(* IEC 61131-3 sources: ATCMcontrol_Engineering/src/Target/ATHW119/Libs/HW119, 8 files *)

(* ---- HW119_CloseCrossTable.st ---- *)
(*[[
    UserText1= "hw119_close_cross_table",
    UserHelpURL= "ATCMfile:HW119_CloseCrossTable.HTML",
]]*)
FUNCTION HW119_CloseCrossTable : UINT
VAR_INPUT
END_VAR
INLINE {STDLIB(HW119_CloseCrossTable)}
END_FUNCTION

(* ---- HW119_dword2float.st ---- *)
(*[[
    UserHelpURL= "ATCMfile:HW119_dword2float.HTML",
    UserText1= "HW119_dword2float",
]]*)
FUNCTION HW119_dword2float : REAL
VAR_INPUT
    dwordvalue : DWORD; (*[dword value to convert]*)
END_VAR
INLINE {STDLIB(HW119_dword2float)}
END_FUNCTION

(* ---- HW119_float2dword.st ---- *)
(*[[
    UserHelpURL= "ATCMfile:HW119_float2dword.HTML",
    UserText1= "HW119_float2dword",
]]*)
FUNCTION HW119_float2dword : DWORD
VAR_INPUT
    realvalue : REAL; (*[float value to convert]*)
END_VAR
INLINE {STDLIB(HW119_float2dword)}
END_FUNCTION

(* ---- HW119_GetAddr.st ---- *)
(*[[
    UserText1= "hw119_get_addr",
    UserHelpURL= "ATCMfile:HW119_GetAddr.HTML",
]]*)
FUNCTION HW119_GetAddr : WORD
VAR_INPUT
    varname : STRING; (*[variable name]*)
END_VAR
INLINE {STDLIB(HW119_GetAddr)}
END_FUNCTION

(* ---- HW119_GetCrossTableField.st ---- *)
(*[[
    UserText1= "hw119_get_cross_table_field",
    UserHelpURL= "ATCMfile:HW119_GetCrossTableField.HTML",
]]*)
FUNCTION HW119_GetCrossTableField : UINT
VAR_INPUT
END_VAR
VAR_OUTPUT
    field : STRING := ''; (*[actual cross table field]*)
END_VAR
INLINE {STDLIB(HW119_GetCrossTableField)}
END_FUNCTION

(* ---- HW119_OpenCrossTable.st ---- *)
(*[[
	UserText1= "hw119_open_cross_table",
    UserHelpURL= "ATCMfile:HW119_OpenCrossTable.HTML",
]]*)
FUNCTION HW119_OpenCrossTable : UINT
VAR_INPUT
    FileName : STRING; (*[cross table file name to open]*)
END_VAR
INLINE {STDLIB(HW119_OpenCrossTable)}
END_FUNCTION

(* ---- HW119_ReadCrossTableRecord.st ---- *)
(*[[
    UserText1= "hw119_read_cross_table_record",
    UserHelpURL= "ATCMfile:HW119_ReadCrossTableRecord.HTML",
]]*)
FUNCTION HW119_ReadCrossTableRecord : UINT
VAR_INPUT
    Alarm : BOOL; (*[set true if it is an alarm or event]*)
END_VAR
INLINE {STDLIB(HW119_ReadCrossTableRecord)}
END_FUNCTION

(* ---- HW119_WriteVar.st ---- *)
(*[[
    UserHelpURL= "ATCMfile:HW119_WriteVar.HTML",
    UserText1= "hw119_write_var",
]]*)
FUNCTION HW119_WriteVar : UINT
VAR_INPUT
    varname : STRING; (*[variable name to write]*)
    value : ANY; (*[value to write]*)
END_VAR

overload STRING(STRING, BOOL)   inline{ EXTLIB((hw119_write_var_bit) }
overload STRING(STRING, BYTE)   inline{ EXTLIB((hw119_write_var_byte) }
overload STRING(STRING, UINT)   inline{ EXTLIB((hw119_write_var_uint) }
overload STRING(STRING, INT)    inline{ EXTLIB((hw119_write_var_int) }
overload STRING(STRING, UDINT)  inline{ EXTLIB((hw119_write_var_udint) }
overload STRING(STRING, DINT)   inline{ EXTLIB((hw119_write_var_dint) }
overload STRING(STRING, REAL)   inline{ EXTLIB((hw119_write_var_real) }
END_FUNCTION
